FUNCTION UpdateEventTimestampWithSystemTime
VAR_INPUT
	stEvent	:	REFERENCE TO ST_Event;
END_VAR
VAR
	fbGETSYSTEMTIME	:	GETSYSTEMTIME;
	
	nTimeLow	:	UDINT;
	nTimeHigh	:	UDINT;
	
	stFileTime	:	T_FILETIME;
END_VAR

fbGETSYSTEMTIME(timeLoDW => stFileTime.dwLowDateTime,
				timeHiDW => stFileTime.dwHighDateTime);
				
stEvent.dtTimestamp := FILETIME_TO_DT(fileTime := stFileTime);

END_FUNCTION

(* stored: Version 1.1.0.1, ProductVersion 3.1.4024.12
   POU UpdateEventTimestampWithSystemTime: Id {7c244887-f4e8-493b-a39e-d0cb95124a33}, SpecialFunc None *)
